INTERFACE I_NciChannel

METHOD BuilDGroup : E_PROGRESS
VAR_INPUT
  Execute           : BOOL;
END_VAR
END_METHOD

PROPERTY CfgAxes : POINTER TO ST_3D_Group
SET
END_SET
END_PROPERTY

PROPERTY ChannelRef : POINTER TO ST_NciChannel_Ref
SET
END_SET
END_PROPERTY

METHOD ClearGroup : E_PROGRESS
VAR_INPUT
  Execute           : BOOL;
END_VAR
END_METHOD

METHOD ConfirmHSK : E_PROGRESS
VAR_INPUT
  Execute           : BOOL;
END_VAR
END_METHOD

METHOD DeleteDistanceToGo : E_PROGRESS
VAR_INPUT
  Execute           : BOOL;
END_VAR
END_METHOD

(*
===============================================================
Error-Flag
===============================================================
*)
PROPERTY Error : BOOL
GET
END_GET
END_PROPERTY

METHOD Error_Get : BOOL
END_METHOD

METHOD EStop : E_PROGRESS
VAR_INPUT
  Execute           : BOOL;
END_VAR
END_METHOD

METHOD GetChannelOverride : real
VAR_INPUT
END_VAR
END_METHOD

METHOD GetItpState : uint
VAR_INPUT
END_VAR
END_METHOD

METHOD GetLoadedProg : string
VAR_INPUT
END_VAR
END_METHOD

(*
===============================================================
Handshake: Announce and acknowledge M-Functions
===============================================================
*)
PROPERTY HSK : BOOL
GET
END_GET
END_PROPERTY

PROPERTY ItpAxes : ST_3D_Group
GET
END_GET
END_PROPERTY

METHOD ItpReset   : E_PROGRESS
VAR_INPUT
  Execute           : BOOL;
END_VAR
END_METHOD

METHOD LoadProg   : E_PROGRESS
VAR_INPUT
  Execute           : BOOL;
END_VAR
END_METHOD

PROPERTY M_FuncReq : word
GET
END_GET
END_PROPERTY

PROPERTY MessageLevel : E_MessageType
SET
END_SET
END_PROPERTY

(*
===============================================================
M-Function
===============================================================
*)
PROPERTY MFunc : INT
GET
END_GET
END_PROPERTY

PROPERTY Override : LREAL
GET
END_GET
SET
END_SET
END_PROPERTY

(*
===============================================================
actual path velo [Units/s]
===============================================================
*)
PROPERTY PathVelo : LREAL
GET
END_GET
END_PROPERTY

(*
===============================================================
G-Code Program Name (sFilePath)
===============================================================
*)
PROPERTY Prog : STRING(255)
GET
END_GET
SET
END_SET
END_PROPERTY

PROPERTY R_ParameterRead : Pointer to ST_R_Parameter;
SET
END_SET
END_PROPERTY

PROPERTY R_ParameterWrite : pointer to ST_R_Parameter;
SET
END_SET
END_PROPERTY

METHOD ReadLine   : E_PROGRESS
VAR_INPUT
  Execute           : BOOL;
END_VAR
//Read G-Code actual Line
VAR_OUTPUT
  ActProgLine       : STRING(100);
END_VAR
END_METHOD

METHOD ReadRParams : E_PROGRESS
VAR_INPUT
  Execute  : BOOL;
END_VAR
END_METHOD

METHOD StartStop : E_PROGRESS
VAR_INPUT
  Execute           : BOOL;
  Start             : BOOL;
  Stop              : BOOL;
END_VAR
END_METHOD

METHOD StepOnAfterEStop : E_PROGRESS
VAR_INPUT
  Execute: BOOL;
END_VAR
END_METHOD

METHOD WriteRParams : E_PROGRESS
VAR_INPUT
  Execute : BOOL;
END_VAR
END_METHOD

END_INTERFACE

(* stored: Version 1.1.0.1, ProductVersion 3.1.4024.12
   Itf I_NciChannel: Id {ef75f316-959e-0835-3611-b097b1464fc3}
   Folder methods: Id {76943757-d4a0-0df4-1a42-45b1dd01bc41}
   Folder properties: Id {bd6dfc2c-2874-0034-396c-573eb0459dae}
   Method BuilDGroup: Id {3e1a0ff4-dc0c-007b-1a25-cbc755c968fd}
   Property CfgAxes: Id {6d0f3be9-a58a-0a3e-269f-25f12935e57b}
   Set Set: Id {a17b3827-ea8b-0a64-13b8-c09d077fde4f}
   Property ChannelRef: Id {36771113-5574-03d7-0084-2394369390e0}
   Set Set: Id {9a93ca84-8c3f-0679-34f1-f6d996690cdd}
   Method ClearGroup: Id {1976b063-c4e7-0102-0e20-a4850da7d26e}
   Method ConfirmHSK: Id {00426d5d-2e6d-0e17-2a36-b622827f55a2}
   Method DeleteDistanceToGo: Id {300c811a-4db2-0b13-09f2-02aa7e70dd91}
   Property Error: Id {55e12491-2b0f-0dc3-107c-da857fb74a4c}
   Get Get: Id {647a9620-a748-0030-316f-b7812eb35c41}
   Method Error_Get: Id {2fdf4a03-72b9-0902-2752-4c88e406c951}
   Method EStop: Id {6c2be89c-2b45-03d5-1f3f-a92d8fd7e29f}
   Method GetChannelOverride: Id {5c31f475-6c13-0035-208c-759f3b2981c8}
   Method GetItpState: Id {a85b3524-f5b5-0d3c-119b-fa1c90864d1b}
   Method GetLoadedProg: Id {43d426f4-cf90-0cf3-3487-4e81f05cd792}
   Property HSK: Id {62d1d256-7ef6-01e7-0eb6-bb78462e5707}
   Get Get: Id {8c061df3-5037-00aa-270f-0cabcd82d737}
   Property ItpAxes: Id {ba8fd14c-0428-0920-1b87-275b99a45ee4}
   Get Get: Id {668d7f56-e2fb-08e2-0e04-0150c9456a17}
   Method ItpReset: Id {08c69477-f264-0bf1-30aa-d08b3e5a417f}
   Method LoadProg: Id {fc827297-3895-09a6-0383-3442c3571958}
   Property M_FuncReq: Id {3304e30a-4e38-0a18-39f8-085b63540fc2}
   Get Get: Id {ffa7ef9b-2860-0015-27d4-bbbcb4f4c69f}
   Property MessageLevel: Id {09df7ffb-d51a-0a46-1af6-e3742a983dbf}
   Set Set: Id {da76445c-8d7c-07d5-2697-cc99925b3ad7}
   Property MFunc: Id {e6813d63-ef99-0544-3d58-efdd02a6e34a}
   Get Get: Id {c2001e49-b3a7-095d-07eb-52c6857e19f5}
   Property Override: Id {076276e8-690e-003b-0b00-b6d1f667a3f4}
   Get Get: Id {e2c3c72b-893f-0af3-1a64-f9a11431c84e}
   Set Set: Id {0d9c029e-0d86-02f1-2b3e-42baf2c0304b}
   Property PathVelo: Id {26d914b0-edd6-0b19-05cc-50e16df7a041}
   Get Get: Id {cd152074-f45b-0b1b-3a3a-2f28700c43c9}
   Property Prog: Id {201ece71-e800-0d84-1292-c36645b1338f}
   Get Get: Id {7663dd05-2dde-05a7-0fb5-757011e98c51}
   Set Set: Id {e844ea91-f14f-0a5b-2b77-80410c5e2627}
   Property R_ParameterRead: Id {a212addd-6c9d-00f3-1a5c-fa995be4af1f}
   Set Set: Id {4cd39b22-d871-03e3-3b5d-ef9d2a33c6a5}
   Property R_ParameterWrite: Id {3526422b-21f0-04a0-1241-28fb5eab3854}
   Set Set: Id {c5a49a41-b4c8-0c83-0c14-68d14dd639db}
   Method ReadLine: Id {b8ab68f8-d791-074f-2c09-4edd328133eb}
   Method ReadRParams: Id {652a9ffe-927d-08aa-0dd4-a63b520763b3}
   Method StartStop: Id {06f443ed-888e-0c1a-0da4-c8532317da42}
   Method StepOnAfterEStop: Id {6154f6bd-15b9-0e13-3e19-4041bf938dc8}
   Method WriteRParams: Id {1fc0647f-ff65-0218-021f-f3649dd685cf} *)
